FUNCTION_BLOCK FB_SequenceControl
VAR_INPUT
	step 					: UDINT;
	stepDescriptionText		: STRING(250);
	logEnableStepInfo		: BOOL;
	logEnableADSLogging		: BOOL;
END_VAR
VAR_OUTPUT
	stepFirstscan 			: BOOL;
	StepActiveTimer 		: TIME;
	ScanCounter 			: ULINT;
	Error					: BOOL;
	ErrorStep				: UDINT;
	LastStepInfo 			: STRING(250);
	NewMessageReady 		: BOOL;
END_VAR
VAR
	stepLast 				: UDINT;
	stepTimer 				: TON;
	LastStepDescriptionText : STRING(250);
	
	StepChangeONS 			: R_TRIG;
	
	StringLength 			: INT;
	StringERRORFind 		: INT;
	StringWARNINGFind 		: INT;
	StringINFORMATIONFind 	: INT;
	Idx 					: INT;
	NewStringTEMP 			: STRING(250);
	NewStringTEMP_Old		: STRING(250);
	DateAndTimeSTRING 		: STRING;
	
	ParsedmessageSTRING		: STRING(250);
	TXTCategory				: INT;
END_VAR

stepTimer(PT := T#24D, ET =>StepActiveTimer);

IF stepLast <> Step THEN
	
	LastStepInfo := CONCAT('Step : ',UDINT_TO_STRING(stepLast));
	
	LastStepInfo := CONCAT(LastStepInfo,' - ');
	LastStepInfo := CONCAT(LastStepInfo,stepDescriptionText);
		
	IF logEnableStepInfo THEN
		IF TIME_TO_DINT(StepActiveTimer) > 0 THEN
			LastStepInfo := 'StepTime : ';
			LastStepInfo := CONCAT(LastStepInfo,TIME_TO_STRING(StepActiveTimer));
		END_IF
		LastStepInfo := CONCAT(LastStepInfo,', ScanCount : ');
		LastStepInfo := CONCAT(LastStepInfo,LINT_TO_STRING(ScanCounter));
	END_IF
		
	stepTimer.IN := 0;
	stepFirstscan := TRUE;
	ScanCounter :=0;
	stepLast := step;
	Error :=0;
	ErrorStep :=0;
	LogNow();
ELSE
	stepFirstscan := FALSE;
	stepTimer.IN := 1;
	NewMessageReady := FALSE;
END_IF

// Timer
ScanCounter := ScanCounter +1;

ACTION LogNow:
NewStringTEMP :='';
StringLength := LEN(stepDescriptionText);						
	IF logEnableADSLogging THEN
		IF StringLength <> 0 THEN
				
			STRINGLENGTH := FIND(stepDescriptionText,'STATUS');
			IF STRINGLENGTH <> 0 THEN
				stepDescriptionText := DELETE(STR:=stepDescriptionText, LEN:=7,POS:=1);
				IF logEnableStepInfo THEN
					stepDescriptionText := CONCAT(stepDescriptionText,' - ');
					stepDescriptionText := CONCAT(stepDescriptionText,LastStepInfo);
				END_IF
				ADSLOGSTR(msgCtrlMask:=ADSLOG_MSGTYPE_LOG , msgFmtStr:=stepDescriptionText , strArg:='' );
			ELSIF STRINGLENGTH <> 0 THEN
		
			STRINGLENGTH := FIND(stepDescriptionText,'ERROR');
				ErrorStep := Step;
				Error := 1;
				stepDescriptionText := DELETE(STR:=stepDescriptionText, LEN:=6,POS:=1);
				IF logEnableStepInfo THEN
					stepDescriptionText := CONCAT(stepDescriptionText,' - ');
					stepDescriptionText := CONCAT(stepDescriptionText,LastStepInfo);
				END_IF
				ADSLOGSTR(msgCtrlMask:=ADSLOG_MSGTYPE_ERROR , msgFmtStr:=ParsedmessageSTRING , strArg:='' );
			ELSIF STRINGLENGTH <> 0 THEN
			
			STRINGLENGTH := FIND(stepDescriptionText,'WARNING');

				stepDescriptionText := DELETE(STR:=stepDescriptionText, LEN:=8,POS:=1);
				IF logEnableStepInfo THEN
					stepDescriptionText := CONCAT(stepDescriptionText,' - ');
					stepDescriptionText := CONCAT(stepDescriptionText,LastStepInfo);
				END_IF
				ADSLOGSTR(msgCtrlMask:=ADSLOG_MSGTYPE_WARN , msgFmtStr:=ParsedmessageSTRING , strArg:='' );
			ELSIF STRINGLENGTH <> 0 THEN

			STRINGLENGTH := FIND(stepDescriptionText,'INFORMATION');

				stepDescriptionText := DELETE(STR:=stepDescriptionText, LEN:=12,POS:=1);
				IF logEnableStepInfo THEN
					stepDescriptionText := CONCAT(stepDescriptionText,' - ');
					stepDescriptionText := CONCAT(stepDescriptionText,LastStepInfo);
				END_IF
				ADSLOGSTR(msgCtrlMask:=ADSLOG_MSGTYPE_LOG , msgFmtStr:=stepDescriptionText , strArg:='' );
			ELSE
				IF logEnableStepInfo THEN
					stepDescriptionText := CONCAT(stepDescriptionText,' - ');
					stepDescriptionText := CONCAT(stepDescriptionText,LastStepInfo);
				END_IF
				ADSLOGSTR(msgCtrlMask:=ADSLOG_MSGTYPE_LOG , msgFmtStr:=stepDescriptionText , strArg:='' );
			END_IF
		END_IF
							
		
	END_IF
	
	IF LastStepDescriptionText <> stepDescriptionText THEN
		NewMessageReady := TRUE;
		LastStepDescriptionText := stepDescriptionText;
	END_IF
END_ACTION

END_FUNCTION_BLOCK

(* stored: Version 1.1.0.1, ProductVersion 3.1.4024.15
   POU FB_SequenceControl: Id {6a52f94b-8522-4a7e-b7a1-e85734f4dc88}, SpecialFunc None
   Action LogNow: Id {eff4a6a9-3618-4480-b636-0cb319ff8534} *)
